(* CODESYS project G42_assignment_1.export

Project tree, tasks and I/O mapping:
  control/
    function block CylinderFB [FBD]
    program cylinder_control_SFC_tsk7 [LD]
    function block LampCTRL [SFC]
    program lamp_ctrl_prg_tsk6 [LD]
    function block Sequence [SFC]
*)

// control/CylinderFB
FUNCTION_BLOCK CylinderFB
VAR_INPUT
	extend: BOOL;
	retract: BOOL;
	cyl_in: BOOL;
	cyl_out: BOOL;
	waitTime: TIME;
END_VAR
VAR_OUTPUT
	ctrl: BOOL;
	count: INT := 0;
	delay: TIME := T#0S;
END_VAR
VAR
	stop: BOOL := FALSE;
	timer: TON;
END_VAR
VAR // added by the converter: edge detectors and wires of the graphical bodies
    _rt1, _rt2 : R_TRIG;
END_VAR

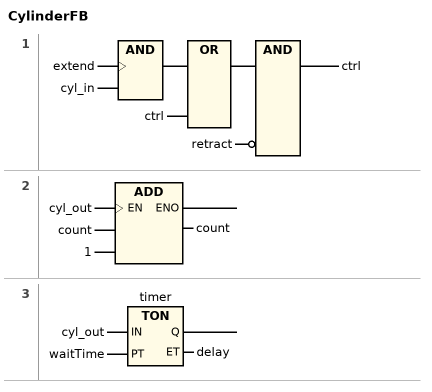
// NETWORK 1
_rt1(CLK := extend);
ctrl := (_rt1.Q AND cyl_in OR ctrl) AND NOT retract;

// NETWORK 2
_rt2(CLK := cyl_out);
IF _rt2.Q THEN count := count + 1; END_IF

// NETWORK 3
timer(IN := cyl_out, PT := waitTime, ET => delay); // TON

END_FUNCTION_BLOCK

// control/cylinder_control_SFC_tsk7
PROGRAM cylinder_control_SFC_tsk7
VAR
	cylinder1: CylinderFB;
	cylinder2: CylinderFB;
	cylinder3: CylinderFB;
	sequence1: Sequence;
END_VAR
VAR // added by the converter: edge detectors and wires of the graphical bodies
    _rt1, _rt2, _rt3 : R_TRIG;
END_VAR

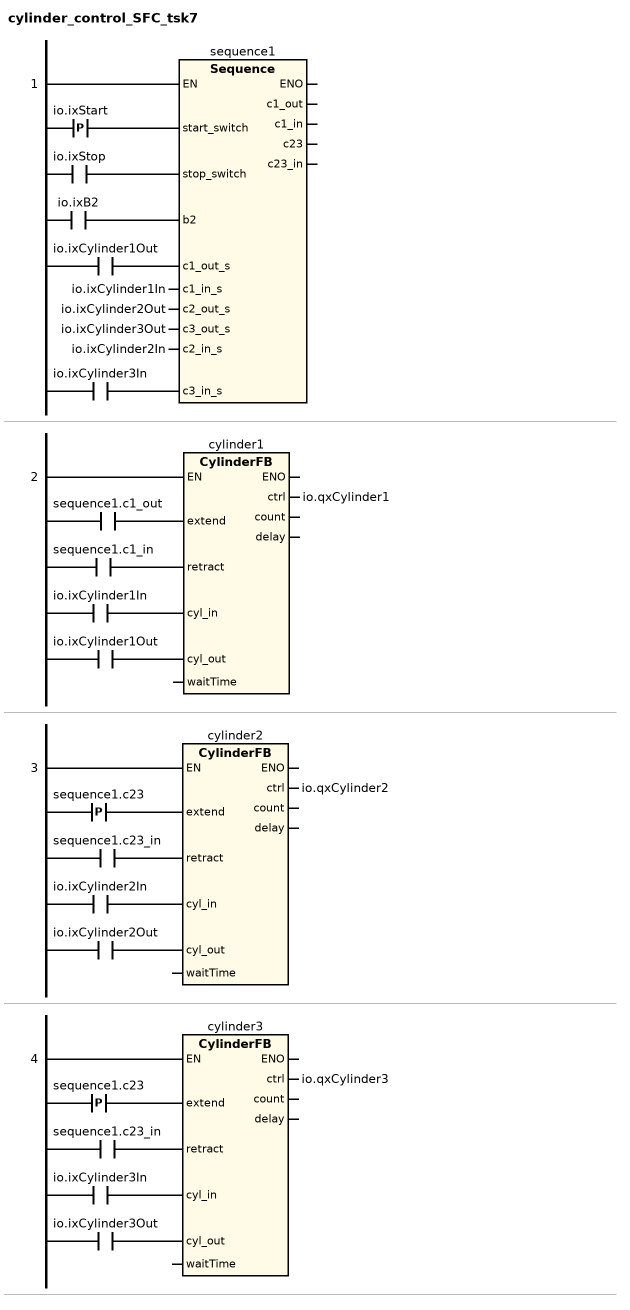
// NETWORK 1
_rt1(CLK := io.ixStart);
sequence1(
    start_switch := _rt1.Q,
    stop_switch := io.ixStop,
    b2 := io.ixB2,
    c1_out_s := io.ixCylinder1Out,
    c1_in_s := io.ixCylinder1In,
    c2_out_s := io.ixCylinder2Out,
    c3_out_s := io.ixCylinder3Out,
    c2_in_s := io.ixCylinder2In,
    c3_in_s := io.ixCylinder3In); // Sequence

// NETWORK 2
cylinder1(
    extend := sequence1.c1_out,
    retract := sequence1.c1_in,
    cyl_in := io.ixCylinder1In,
    cyl_out := io.ixCylinder1Out,
    ctrl => io.qxCylinder1); // CylinderFB

// NETWORK 3
_rt2(CLK := sequence1.c23);
cylinder2(
    extend := _rt2.Q,
    retract := sequence1.c23_in,
    cyl_in := io.ixCylinder2In,
    cyl_out := io.ixCylinder2Out,
    ctrl => io.qxCylinder2); // CylinderFB

// NETWORK 4
_rt3(CLK := sequence1.c23);
cylinder3(
    extend := _rt3.Q,
    retract := sequence1.c23_in,
    cyl_in := io.ixCylinder3In,
    cyl_out := io.ixCylinder3Out,
    ctrl => io.qxCylinder3); // CylinderFB

END_PROGRAM

// control/Sequence
FUNCTION_BLOCK Sequence
VAR_INPUT
	start_switch: BOOL;
	stop_switch: BOOL;
	b2:BOOL;
	c1_out_s:BOOL;
	c1_in_s: BOOL;
	c2_out_s: BOOL;
	c3_out_s: BOOL;
	c2_in_s: BOOL;
	c3_in_s: BOOL;
END_VAR
VAR_OUTPUT
	c1_out:BOOL;
	c1_in:BOOL;
	c23:BOOL;
	c23_in: BOOL;
END_VAR
VAR
END_VAR

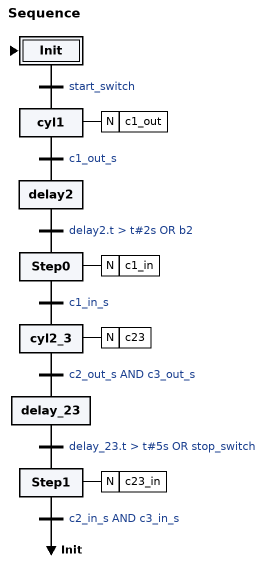
INITIAL_STEP Init:
END_STEP
TRANSITION FROM Init TO cyl1
    := start_switch;
END_TRANSITION
STEP cyl1:
    c1_out(N);
END_STEP
TRANSITION FROM cyl1 TO delay2
    := c1_out_s;
END_TRANSITION
STEP delay2:
END_STEP
TRANSITION FROM delay2 TO Step0
    := delay2.t > t#2s OR b2;
END_TRANSITION
STEP Step0:
    c1_in(N);
END_STEP
TRANSITION FROM Step0 TO cyl2_3
    := c1_in_s;
END_TRANSITION
STEP cyl2_3:
    c23(N);
END_STEP
TRANSITION FROM cyl2_3 TO delay_23
    := c2_out_s AND c3_out_s;
END_TRANSITION
STEP delay_23:
END_STEP
TRANSITION FROM delay_23 TO Step1
    := delay_23.t > t#5s OR stop_switch;
END_TRANSITION
STEP Step1:
    c23_in(N);
END_STEP
TRANSITION FROM Step1 TO Init
    := c2_in_s AND c3_in_s;
END_TRANSITION

END_FUNCTION_BLOCK

// control/LampCTRL
FUNCTION_BLOCK LampCTRL
VAR_INPUT
	 start: BOOL;
	 start_switch: BOOL;
END_VAR
VAR_OUTPUT
	l1: BOOL;
	l2: BOOL;
	l3: BOOL;
	l4: BOOL;
END_VAR
VAR
END_VAR

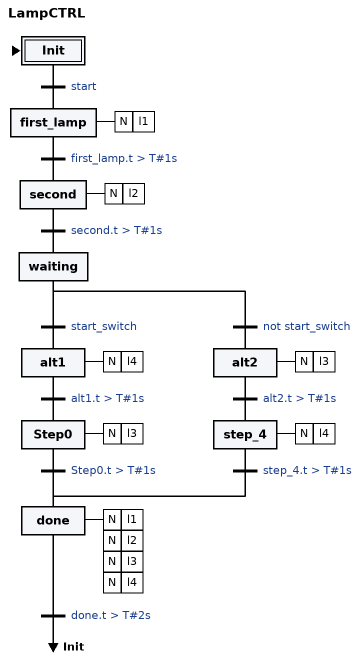
INITIAL_STEP Init:
END_STEP
TRANSITION FROM Init TO first_lamp
    := start;
END_TRANSITION
STEP first_lamp:
    l1(N);
END_STEP
TRANSITION FROM first_lamp TO second
    := first_lamp.t > T#1s;
END_TRANSITION
STEP second:
    l2(N);
END_STEP
TRANSITION FROM second TO waiting
    := second.t > T#1s;
END_TRANSITION
STEP waiting:
END_STEP
TRANSITION FROM waiting TO alt1
    := start_switch;
END_TRANSITION
STEP alt1:
    l4(N);
END_STEP
TRANSITION FROM alt1 TO Step0
    := alt1.t > T#1s;
END_TRANSITION
STEP Step0:
    l3(N);
END_STEP
TRANSITION FROM Step0 TO done
    := Step0.t > T#1s;
END_TRANSITION
TRANSITION FROM waiting TO alt2
    := not start_switch;
END_TRANSITION
STEP alt2:
    l3(N);
END_STEP
TRANSITION FROM alt2 TO step_4
    := alt2.t > T#1s;
END_TRANSITION
STEP step_4:
    l4(N);
END_STEP
TRANSITION FROM step_4 TO done
    := step_4.t > T#1s;
END_TRANSITION
STEP done:
    l1(N);
    l2(N);
    l3(N);
    l4(N);
END_STEP
TRANSITION FROM done TO Init
    := done.t > T#2s;
END_TRANSITION

END_FUNCTION_BLOCK

// control/lamp_ctrl_prg_tsk6
PROGRAM lamp_ctrl_prg_tsk6
VAR
	lamp_testing: LampCTRL;
END_VAR

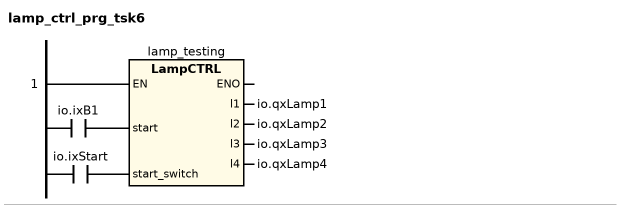
// NETWORK 1
lamp_testing(
    start := io.ixB1,
    start_switch := io.ixStart,
    l1 => io.qxLamp1,
    l2 => io.qxLamp2,
    l3 => io.qxLamp3,
    l4 => io.qxLamp4); // LampCTRL

END_PROGRAM
